Fanuc KAREL source: kt00493.KL

-- PROVISIONAL review KL for V770-1; original PC SHA256 dbc1addc7f72804b50984ee59848dc0915fd22a2e253c339e39ea64502033fe4
-- Incomplete behavior may be omitted. Consult companion uncertainty JSON. Do not deploy.
PROGRAM KT00493
%NOLOCKGROUP
VAR
  OUT : BOOLEAN
-- UNRESOLVED_DECL P1 type=000102
-- UNRESOLVED_DECL P2 type=000101
BEGIN
  -- UNRESOLVED_PC offsets 5-20; opcodes 2E,22,32,35
  -- UNRESOLVED_PC offsets 25-53; opcodes 49,7E,49,AC,23
  -- UNRESOLVED_PC offsets 58-62; opcodes 7F
END KT00493
